FUNCTION_BLOCK FB_SplitWordToByte
////////////////// 
// Convert one REAL into  2 separate WORDS in Big Endian Encoding. 
//////////////////	
VAR_INPUT
	IN		: WORD ;				// Real input
	
END_VAR

VAR_OUTPUT
	STRONG_BYTE		: BYTE;	// Word output array
	WEAK_BYTE		: BYTE;	// Word output array
END_VAR

STRONG_BYTE := WORD_TO_BYTE(IN) ; 				
WEAK_BYTE 	:= WORD_TO_BYTE(SHR(IN,8));

END_FUNCTION_BLOCK

(* stored: Version 1.1.0.1, ProductVersion 3.1.4024.6
   POU FB_SplitWordToByte: Id {acac4b2c-b0d3-458f-8789-8b9d4f8e8ce9}, SpecialFunc None *)
